Omron CX-Programmer project NewProject (CX-Programmer 9.75)

# PLC NewPLC1: CJ2M CPU11

## Global symbols (name address type ; comment)
0.01 BOOL  ; START
0.02 BOOL  ; STOP
0.03 BOOL  ; SWITCH1
0.04 BOOL  ; SWITCH2
0.05 BOOL  ; SWITCH3
1.00 BOOL  ; RUN
1.01 BOOL  ; MOTOR1
1.02 BOOL  ; MOTOR2
1.03 BOOL  ; MOTOR3

## Program INDUSTRIAL_AUTOMATION_PLC_PROGRAMMING (cyclic task 0)
; CONVEYOR BELT SERIES MOTOR CONTROL

### Section RUNG_SETUP
; LADDER LOGIC PROGRAMMING OMRON PLC

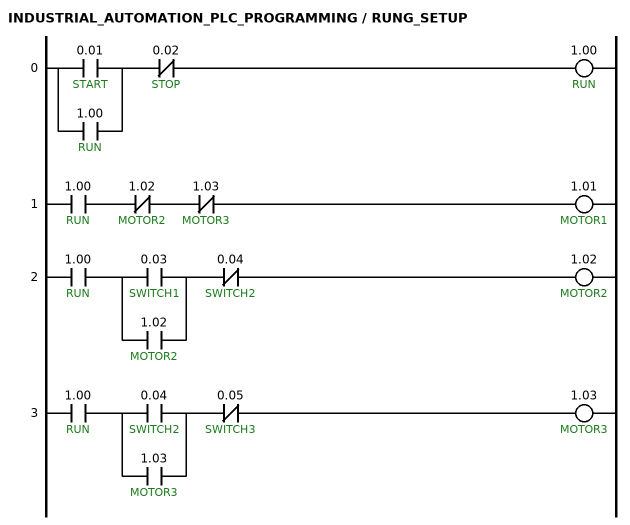
; rung 0
LD 0.01  ; START
OR 1.00  ; RUN
ANDNOT 0.02  ; STOP
OUT 1.00  ; RUN
; rung 1
LD 1.00  ; RUN
ANDNOT 1.02  ; MOTOR2
ANDNOT 1.03  ; MOTOR3
OUT 1.01  ; MOTOR1
; rung 2
LD 1.00  ; RUN
LD 0.03  ; SWITCH1
OR 1.02  ; MOTOR2
ANDLD
ANDNOT 0.04  ; SWITCH2
OUT 1.02  ; MOTOR2
; rung 3
LD 1.00  ; RUN
LD 0.04  ; SWITCH2
OR 1.03  ; MOTOR3
ANDLD
ANDNOT 0.05  ; SWITCH3
OUT 1.03  ; MOTOR3

### Section END
; rung 0
END(001)